FUNCTION_BLOCK wifi (* Service Interface Function Block Type *)
  (* Standard: 61499-2; Description: Copyright (c) 2026 HR Agrartechnik GmbH This program and the accompanying materials are made available under the terms of the Eclipse Public License 2.0 which is available at https://www.eclipse.org/legal/epl-2.0/ SPDX-License-Identifier: EPL-2.0 *)
  (* Version 1.0, 2025-07-09, Franz Höpfinger, HR Agrartechnik GmbH *)
  IMPORT eclipse4diac::core::TypeHash;
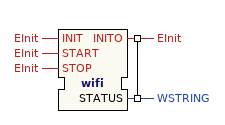
  EVENT_INPUT
    INIT : EInit; (* Service Initialization *)
    START : EInit; (* Start WiFi *)
    STOP : EInit; (* Stop WiFi *)
  END_EVENT
  EVENT_OUTPUT
    INITO : EInit WITH STATUS; (* Initialization Confirm *)
  END_EVENT
  VAR_OUTPUT
    STATUS : WSTRING; (* Service Status *)
  END_VAR
END_FUNCTION_BLOCK
